(* PLC project Unnamed, Unknown Unnamed 1 *)
(* stored: creationDateTime 2025-04-10T09:55:54, modificationDateTime 2025-04-10T10:11:42 *)

PROGRAM program0
  VAR
    StartButton : BOOL;
    StopButton : BOOL;
    Motor : BOOL;
  END_VAR

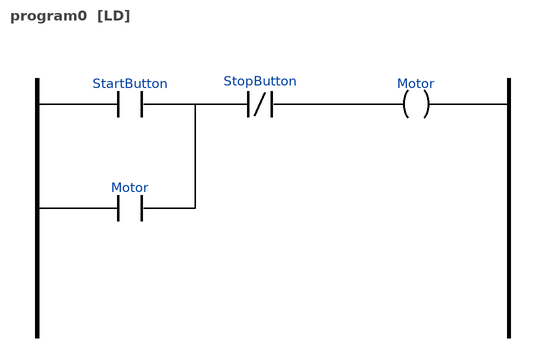
(* LD diagram, written out as Structured Text *)
Motor := (StartButton OR Motor) AND NOT StopButton;
END_PROGRAM

CONFIGURATION Config0
  RESOURCE Res0 ON PLC
    TASK task0(INTERVAL := T#20ms, PRIORITY := 0);
    PROGRAM instance0 WITH task0 : program0;
  END_RESOURCE
END_CONFIGURATION
